{attribute 'GeneratedUsingTerminal: EK1122-0000-0018'}
{attribute addProperty BoxType "EK1122-0000-0018"}
{attribute addProperty Id "Term_17_EK1100Term_17_EK1100_34C4A2BF164"}
{attribute addProperty CRC "3413821643"}
{attribute addProperty Size "164"}
TYPE Term_16_EK1122_CB7AC8CB EXTENDS EK1122_2A90D53A :
STRUCT
	{attribute addProperty Name "Term_17_EK1100"}
	{attribute addProperty PreviousPort "Term 16 (EK1122) : D"}
	Term_17_EK1100 : Term_17_EK1100_34C4A2BF;
END_STRUCT
END_TYPE

(* stored: Version 1.2.0.0, ProductVersion 3.1.4024.9
   DUT Term_16_EK1122_CB7AC8CB: Id {e1256a89-881a-08fa-337a-b6bdcbb33117} *)
